// TIA Portal V17 export
// export: Created 2024-08-09T12:50:43.7435413Z, ExportSetting WithDefaults, DisplayName Totally Integrated Automation Portal, DisplayVersion V17 Update 7, DisplayName TIA Portal Openness, DisplayVersion V17 Update 7, DisplayName TIA Portal Version Control Interface, DisplayVersion V17, DisplayName STEP 7 Professional, DisplayVersion V17 Update 7, DisplayName STEP 7 Safety, DisplayVersion V17 Update 6, DisplayName WinCC Professional, DisplayVersion V17 Update 7
DATA_BLOCK "idbSql4Siemens"   // DB1000
VERSION : 0.1
// stored: AutoNumber false, DBAccessibleFromOPCUA true, DBAccessibleFromWebserver true, InstanceOfName fbSql4Siemens, InstanceOfType FB
"fbSql4Siemens"
   // VAR_INPUT
   //    iIP1 : Int;
   //    iIP2 : Int;
   //    iIP3 : Int;
   //    iIP4 : Int;
   //    iRemotePort : Int;
   //    iLocalPort : Int;
   //    tTimeout : Time;
   //    iConnectionID : CONN_OUC;
   //    wHardwareID : HW_ANY;
   //    tFbExecTimeLimit : Time;
   // END_VAR
   // VAR_OUTPUT
   //    tFbExecTimeMax : Time;
   //    tLastRequest : Time;
   // END_VAR
   // VAR_IN_OUT
   //    stSql4SiemensInterface : "utSql4SiemensInterface";
   // END_VAR
   // VAR
   //    stTcpV4 { S7_SetPoint := 'True'} : TCON_IP_v4;
   //    inTsendC { S7_SetPoint := 'True'} : TSEND_C;
   //    inTrcv { S7_SetPoint := 'True'} : TRCV;
   //    xTsendReq { ExternalVisible := 'False'} : Bool;
   //    xTsendCont : Bool;
   //    xTsendDone { ExternalVisible := 'False'} : Bool;
   //    xTsendBusy { ExternalVisible := 'False'} : Bool;
   //    xTsendError { ExternalVisible := 'False'} : Bool;
   //    wTsendState { ExternalVisible := 'False'} : Word;
   //    xTrcvEnR : Bool;
   //    xTrcvNdr : Bool;
   //    xTrcvBusy : Bool;
   //    xTrcvError : Bool;
   //    wTrcvState { ExternalVisible := 'False'} : Word;
   //    udiTrcvLen { ExternalVisible := 'False'} : UDInt;
   //    iStep : Int;
   //    inTimeout { S7_SetPoint := 'True'} : TON_TIME;
   //    xTimeout { ExternalVisible := 'False'} : Bool;
   //    inExecuteTimeout { S7_SetPoint := 'True'} : TON_TIME;
   //    abRcvData { ExternalVisible := 'False'} : Array[0..5999] of Byte;
   //    diRow : DInt;
   //    diCol : DInt;
   //    diPos : DInt;
   //    diNewPos : DInt;
   //    tRequestStart : DTL;
   //    xResponseDone : Bool;
   //    sValue : WString[300];
   //    diResultState_S : DInt;
   //    diResultReturnParams_S : DInt;
   //    diResultRows_S : DInt;
   //    diResultCols_S : DInt;
   //    tFbExecTimeMax_S : Time;
   // END_VAR
BEGIN
END_DATA_BLOCK
